PROGRAM PRG_PID_CALL
VAR
	
END_VAR




// C3 EL3024 Channel 3 analog 4-20mA from thermocouple range 0-32767
// Measure -40F to 140F
GVL_IO.rAIInput3 := (Thermocouple/(32767.0 - 0.0))* 100;

HeaterOnRequest := PRG_FB_CTRL_PID.fOut;
PRG_FB_CTRL_PID();

//Call simulated PID for debugging locally. Comment out after commissioning
//PRG_SIM_PROCESS();

END_PROGRAM

(* stored: Version 1.1.0.1, ProductVersion 3.1.4024.12
   POU PRG_PID_CALL: Id {92b1ff5d-55bb-49fa-97be-bafe0d32ba6a}, SpecialFunc None *)
